// TIA Portal V19 export
FUNCTION_BLOCK "Painting_Chamber"   // FB4, LAD
{ S7_Optimized_Access := 'TRUE' }
// stored: MemoryReserve 100, SetENOAutomatically false
   VAR_INPUT
      Sensor_102B5 : Bool;
      Sensor_102B6 : Bool;
      Open_Valve : Bool;
   END_VAR
   VAR_OUTPUT
      Valve_106Q6 : Bool;
      Motor_4Q5 : Bool;
   END_VAR
   VAR
      Motor_Control : Bool;
   END_VAR
   VAR_TEMP   // added for the SCL form of the ladder/FBD networks
      _w1 : Bool;
   END_VAR
BEGIN

REGION Network 1
   // V 0.1.1 Updated connection for motor
   // V 0.1.0 Preliminary sketch
   // Connection for OnOff_regulator
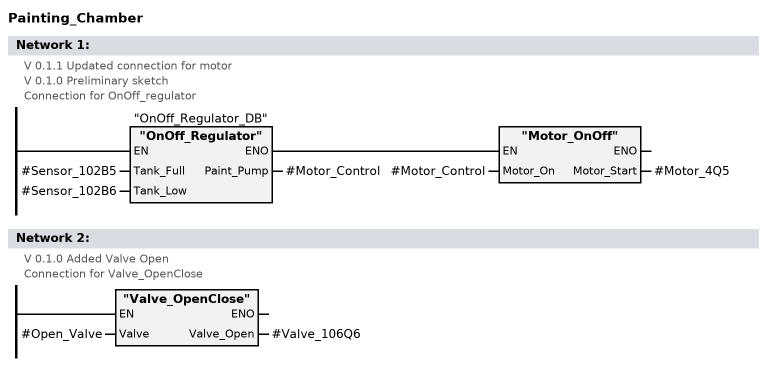
   RUNG wire#powerrail
      "OnOff_Regulator_DB"(Tank_Full := #Sensor_102B5, Tank_Low := #Sensor_102B6, Paint_Pump => #Motor_Control)
      "Motor_OnOff"(Motor_On := #Motor_Control, Motor_Start => #Motor_4Q5)
   END_RUNG
   // the same network as SCL:
   "OnOff_Regulator_DB"(Tank_Full := #Sensor_102B5,   // "OnOff_Regulator"
                        Tank_Low := #Sensor_102B6,
                        Paint_Pump => #Motor_Control,
                        ENO => #_w1);
   IF #_w1 THEN "Motor_OnOff"(Motor_On := #Motor_Control, Motor_Start => #Motor_4Q5); END_IF;
END_REGION

REGION Network 2
   // V 0.1.0 Added Valve Open
   // Connection for Valve_OpenClose
   RUNG wire#powerrail
      "Valve_OpenClose"(Valve := #Open_Valve, Valve_Open => #Valve_106Q6)
   END_RUNG
   // the same network as SCL:
   "Valve_OpenClose"(Valve := #Open_Valve, Valve_Open => #Valve_106Q6);
END_REGION
END_FUNCTION_BLOCK
